// A bit of comment
TYPE SystemParametersXXL :
STRUCT
	Operation: SystemOperationParametersXXL;
END_STRUCT
END_TYPE

(* stored: Version 1.1.0.1, ProductVersion 3.1.4024.6
   DUT SystemParametersXXL: Id {3dae6fd6-0e2c-48fd-a262-a277eaa45759} *)
